(* IEC 61131-3 sources: com.logicals.lc3.webinar/usRTS_RPMControl_iSOC/src_FB_LIB_SAFE/Counter/LINT, 3 files *)

(* ---- wCTD_LINT.iecst ---- *)
NAMESPACE logicals.web.standard
NAMESPACE counter

/*
 * Function block wrapper for IEC 61131-3 CTD_LINT<br>
 * CD = decrement on positive edge on CD (BOOL)<br>
 * LD = flag for reset (CV:=PV) (BOOL)<br>
 * PV = initial value for counting (LINT)<br>
 * Q  = flag showing whether 0 is reached or not (BOOL)<br>
 * CV = current value of counter (LINT)<br>
 */
FUNCTION_BLOCK wCTD_LINT
	{ CV { index := 2 }; vNameAlignment:="center"; altName:="CTD_LINT"; bgColor:="LightPink"; width:=120; }
	VAR_INPUT
		CD : BOOL /* R_EDGE */;
		LD : BOOL;
		PV : LINT;
	END_VAR
	VAR_OUTPUT
		Q  : BOOL;
		CV : LINT;
	END_VAR
	VAR
		CTD_LINT : CTD_LINT;
	END_VAR

	CTD_LINT(CD:=CD, LD:=LD, PV:=PV, Q=>Q, CV=>CV, ENO=>ENO);
END_FUNCTION_BLOCK

END_NAMESPACE
END_NAMESPACE

(* ---- wCTU_LINT.iecst ---- *)
NAMESPACE logicals.web.standard
NAMESPACE counter

/*
 * Function block wrapper for IEC 61131-3 CTU_LINT<br>
 * CU = increment on positive edge on CU (BOOL)<br>
 * R  = flag for reset (BOOL)<br>
 * PV = upper limit of counter (LINT)<br>
 * Q  = flag showing whether upper limit is reached or not (BOOL)<br>
 * CV = current value of counter (LINT)<br>
 */
FUNCTION_BLOCK wCTU_LINT
	{ CV { index := 2 }; vNameAlignment:="center"; altName:="CTU_LINT"; bgColor:="LightPink"; width:=120; }
	VAR_INPUT
		CU : BOOL /* R_EDGE */;
		R  : BOOL;
		PV : LINT;
	END_VAR
	VAR_OUTPUT
		Q  : BOOL;
		CV : LINT;
	END_VAR
	VAR
		M : BOOL;
	END_VAR
	VAR_TEMP
		edgeCU : BOOL;
	END_VAR

	/* Perform Edge Recognition */
	IF CU THEN
		edgeCU := NOT M;
		M := TRUE;
	ELSE
		edgeCU := CU;
		M := FALSE;
	END_IF;

	IF R THEN
		CV := 0;
	ELSE
		IF edgeCU THEN
			IF CV < 16#7FFFFFFFFFFFFFFF THEN
				CV := CV + 1;
			END_IF;
		END_IF;
	END_IF;
	Q := CV >= PV;
END_FUNCTION_BLOCK

END_NAMESPACE
END_NAMESPACE

(* ---- wCTUD_LINT.iecst ---- *)
NAMESPACE logicals.web.standard
NAMESPACE counter

/*
 * Function block wrapper for IEC 61131-3 CTUD_LINT<br>
 * CU = increment on positive edge on CU (BOOL)<br>
 * CD = decrement on positive edge on CD (BOOL)<br>
 * R  = flag for reset (CV:=0) (BOOL)<br>
 * LD = flag for load (CV:=PV) (BOOL)<br>
 * PV = upper limit of counter (LINT)<br>
 * QU = flag showing whether upper limit is reached or not (BOOL)<br>
 * QD = flag showing whether 0 is reached or not (BOOL)<br>
 * CV = current value of counter (LINT)<br>
 */
FUNCTION_BLOCK wCTUD_LINT
	{ vNameAlignment:="center"; altName:="CTUD_LINT"; bgColor:="LightPink"; width:=120; }
	VAR_INPUT
		CU : BOOL /* R_EDGE */;
		CD : BOOL /* R_EDGE */;
		R  : BOOL;
		LD : BOOL;
		PV : LINT;
	END_VAR
	VAR_OUTPUT
		QU : BOOL;
		QD : BOOL;
		CV : LINT;
	END_VAR
	VAR
		CTUD_LINT : CTUD_LINT;
	END_VAR

	CTUD_LINT(CU:=CU, CD:=CD, R:=R, LD:=LD, PV:=PV, QU=>QU, QD=>QD, CV=>CV, ENO=>ENO);
END_FUNCTION_BLOCK

END_NAMESPACE
END_NAMESPACE
